// TIA Portal V20 export
TYPE "UDT_MTP_AnaView"
TITLE = MTPDataObjectSUCLibrary/DataAssembly/AnaView
   STRUCT
      VSclMin { ExternalWritable := 'False'} : Real := 0.0;   // Value Scale Low Limit
      VSclMax { ExternalWritable := 'False'} : Real := 100.0;   // Value Scale High Limit
      VUnit { ExternalWritable := 'False'} : Int := 1001;   // Value Unit
      OSLevel : Byte := 16#00;   // OSLevel variable
      WQC { ExternalWritable := 'False'} : Byte := 16#FF;   // Worst Quality code
      V { ExternalWritable := 'False'} : Real := 0.0;   // Value
   END_STRUCT;
END_TYPE
